// TIA Portal V16 export
// export: Created 2021-08-30T10:49:32.4865879Z, ExportSetting WithDefaults, DisplayName Totally Integrated Automation Portal, DisplayVersion V16 Update 3, DisplayName TIA Portal Version Control Interface, DisplayVersion V16 Update 2, DisplayName TIA Portal Openness, DisplayVersion V16 Update 3, DisplayName TIA Portal Teamcenter Gateway, DisplayVersion V16, DisplayName STEP 7 Professional, DisplayVersion V16 Update 3, DisplayName STEP 7 Safety, DisplayVersion V16, DisplayName WinCC Advanced, DisplayVersion V16 Update 3
FUNCTION_BLOCK "PumpCntrl2Pu1Fc"   // FB61, FBD
{ S7_Optimized_Access := 'TRUE' }
VERSION : 0.1
// 0 0 -стоп, 1- работа
// 1 2 - Запуск
// 2 4 - Остановка
// 3 8 - Сервисный режим
// 4 16 - Ошибка пуска
// 5 32 - Ошибка останова
// 6 64 - Ошибка питания
// 7 128 - Ошибка Частотника
// 8 256 - Блокировка внешняя (сборная)
// 9 - 512 - Нажат аварийный стоп
// 10 -U24 - Сборная авария
// 11 - 2048 - Местный режим
// 12 -  4096 - Ошибка вклчюния контактора
// 13 - 8192 - шбика отключения контактора
// 14 -  16384 - 1 показывать кнопки ручного управления
// 15 - 32768 - режим 1-ручной, 0-авто (только для индикатора на скаде)
// stored: AutoNumber false, IsIECCheckEnabled false, IsRetainMemResEnabled false, MemoryReserve 100, SetENOAutomatically false, UDAEnableTagReadback false
   VAR_INPUT
      modePU : Bool;
      cmPU : Bool;
      iWorkUZ : Bool;
      iAlarmFC : Bool;
      iKM1 : Bool;
      iKM2 : Bool;
      enableChange : Bool;
      Ack : Bool;
      blockPU1_1 : Bool;
      blockPU1_2 : Bool;
      blockPU1_3 : Bool;
      blockPU1_4 : Bool;
      blockPU1_5 : Bool;
      blockPU1_6 : Bool;
      blockPU1_7 : Bool;
      blockPU1_8 : Bool;
      blockPU2_1 : Bool;
      blockPU2_2 : Bool;
      blockPU2_3 : Bool;
      blockPU2_4 : Bool;
      blockPU2_5 : Bool;
      blockPU2_6 : Bool;
      blockPU2_7 : Bool;
      blockPU2_8 : Bool;
   END_VAR
   VAR_OUTPUT
      qKM_PU1 : Bool;
      qKM_PU2 : Bool;
      qUZ : Bool;
      showPU1_button : Bool;
      showPU2_button : Bool;
      tChangeRealHour : Real;
   END_VAR
   VAR_IN_OUT
      select : Bool;
      PU1 : "Pump";
      PU2 : "Pump";
   END_VAR
   VAR
      cmPU1 : Bool;   // Врутренняя команда первого насоса
      cmPU2 : Bool;   // Врутренняя команда второго насоса
      selectInternal : Bool;
      TOFcmPU1 { S7_SetPoint := 'True'} : TOF_TIME;
      TOFcmPU2 { S7_SetPoint := 'True'} : TOF_TIME;
   END_VAR
   VAR RETAIN
      tWork1 : DInt;
      tWork2 : DInt;
   END_VAR
   VAR
      tChange : DInt;
      needChange : Bool;
      tmpDInt : DInt;
      errAlarmFC_PU1 : Bool;
      errAlarmFC_PU2 : Bool;
      errBlock_PU1 : Bool;
      errBlock_PU2 : Bool;
      tmrErrOnUZ : TON_TIME;
      errON_UZ_PU1 : Bool;
      errON_UZ_PU2 : Bool;
      tmrErrOffUZ : TON_TIME;
      errOff_UZ_PU1 : Bool;
      errOff_UZ_PU2 : Bool;
      tmrErrOnKM_PU1 : TON_TIME;
      errOn_KM_PU1 : Bool;
      errOn_KM_PU2 : Bool;
      errOff_KM_PU1 : Bool;
      errOff_KM_PU2 : Bool;
      tmrErrOnKM_PU2 { S7_SetPoint := 'True'} : TON_TIME;
      tmrErrOffKM_PU1 { S7_SetPoint := 'True'} : TON_TIME;
      tmrErrOffKM_PU2 { S7_SetPoint := 'True'} : TON_TIME;
      errServicePU1 : Bool;
      errServicePU2 : Bool;
      tStartPU_FC : Time;
      tStopPU_FC : Time;
   END_VAR
BEGIN

REGION Network 1: Режим
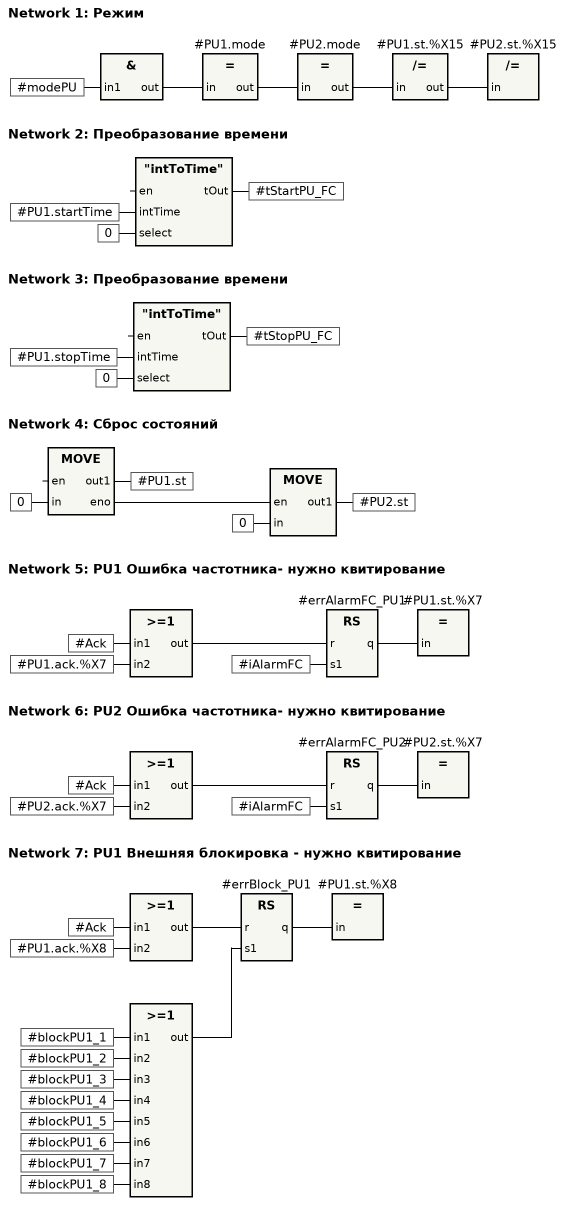
   #PU1.mode := #modePU;
   #PU2.mode := #modePU;
   #PU1.st.%X15 := NOT #modePU;
   #PU2.st.%X15 := NOT #modePU;
END_REGION

REGION Network 2: Преобразование времени
   // ВРемя из настроек первого насоса
   "intToTime"(intTime := #PU1.startTime, select := 0, tOut => #tStartPU_FC);
END_REGION

REGION Network 3: Преобразование времени
   // ВРемя из настроек первого насоса
   "intToTime"(intTime := #PU1.stopTime, select := 0, tOut => #tStopPU_FC);
END_REGION

REGION Network 4: Сброс состояний
   #PU1.st := 0;
   #PU2.st := 0;
END_REGION

REGION Network 5: PU1 Ошибка частотника- нужно квитирование
   IF #Ack OR #PU1.ack.%X7 THEN
       #errAlarmFC_PU1 := FALSE;   // RS flip-flop
   END_IF;
   IF #iAlarmFC THEN #errAlarmFC_PU1 := TRUE; END_IF;
   #PU1.st.%X7 := #errAlarmFC_PU1;
END_REGION

REGION Network 6: PU2 Ошибка частотника- нужно квитирование
   IF #Ack OR #PU2.ack.%X7 THEN
       #errAlarmFC_PU2 := FALSE;   // RS flip-flop
   END_IF;
   IF #iAlarmFC THEN #errAlarmFC_PU2 := TRUE; END_IF;
   #PU2.st.%X7 := #errAlarmFC_PU2;
END_REGION

REGION Network 7: PU1 Внешняя блокировка - нужно квитирование
   IF #Ack OR #PU1.ack.%X8 THEN
       #errBlock_PU1 := FALSE;   // RS flip-flop
   END_IF;
   IF #blockPU1_1 OR #blockPU1_2 OR #blockPU1_3 OR #blockPU1_4 OR #blockPU1_5 OR #blockPU1_6 OR #blockPU1_7 OR #blockPU1_8 THEN
       #errBlock_PU1 := TRUE;
   END_IF;
   #PU1.st.%X8 := #errBlock_PU1;
END_REGION

REGION Network 8: Детализация блокировок PU1
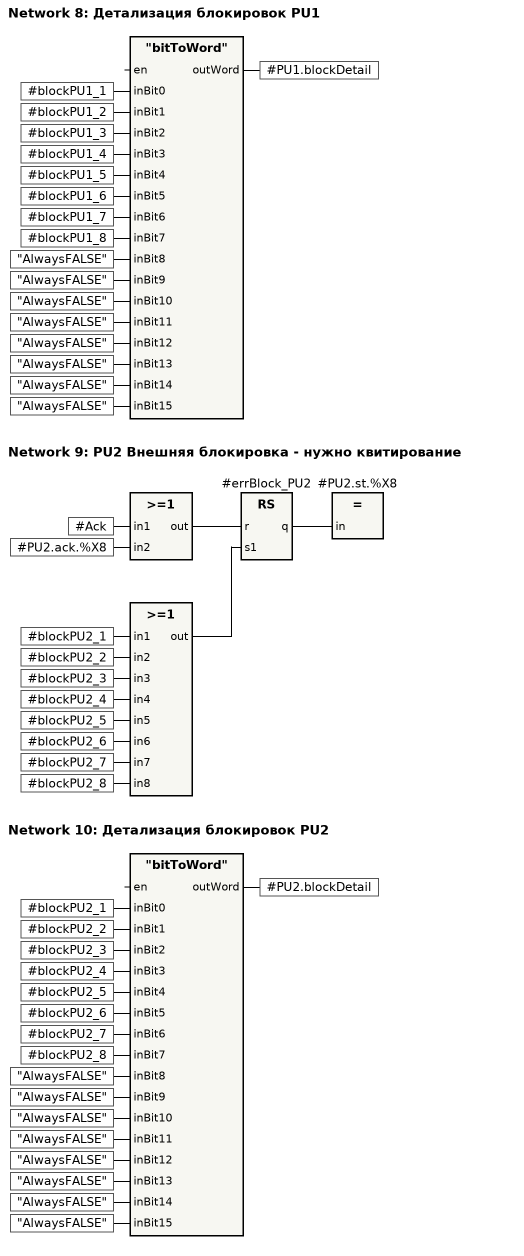
   "bitToWord"(inBit0 := #blockPU1_1,
               inBit1 := #blockPU1_2,
               inBit2 := #blockPU1_3,
               inBit3 := #blockPU1_4,
               inBit4 := #blockPU1_5,
               inBit5 := #blockPU1_6,
               inBit6 := #blockPU1_7,
               inBit7 := #blockPU1_8,
               inBit8 := "AlwaysFALSE",
               inBit9 := "AlwaysFALSE",
               inBit10 := "AlwaysFALSE",
               inBit11 := "AlwaysFALSE",
               inBit12 := "AlwaysFALSE",
               inBit13 := "AlwaysFALSE",
               inBit14 := "AlwaysFALSE",
               inBit15 := "AlwaysFALSE",
               outWord => #PU1.blockDetail);
END_REGION

REGION Network 9: PU2 Внешняя блокировка - нужно квитирование
   IF #Ack OR #PU2.ack.%X8 THEN
       #errBlock_PU2 := FALSE;   // RS flip-flop
   END_IF;
   IF #blockPU2_1 OR #blockPU2_2 OR #blockPU2_3 OR #blockPU2_4 OR #blockPU2_5 OR #blockPU2_6 OR #blockPU2_7 OR #blockPU2_8 THEN
       #errBlock_PU2 := TRUE;
   END_IF;
   #PU2.st.%X8 := #errBlock_PU2;
END_REGION

REGION Network 10: Детализация блокировок PU2
   "bitToWord"(inBit0 := #blockPU2_1,
               inBit1 := #blockPU2_2,
               inBit2 := #blockPU2_3,
               inBit3 := #blockPU2_4,
               inBit4 := #blockPU2_5,
               inBit5 := #blockPU2_6,
               inBit6 := #blockPU2_7,
               inBit7 := #blockPU2_8,
               inBit8 := "AlwaysFALSE",
               inBit9 := "AlwaysFALSE",
               inBit10 := "AlwaysFALSE",
               inBit11 := "AlwaysFALSE",
               inBit12 := "AlwaysFALSE",
               inBit13 := "AlwaysFALSE",
               inBit14 := "AlwaysFALSE",
               inBit15 := "AlwaysFALSE",
               outWord => #PU2.blockDetail);
END_REGION

REGION Network 11: таймер включения частотника
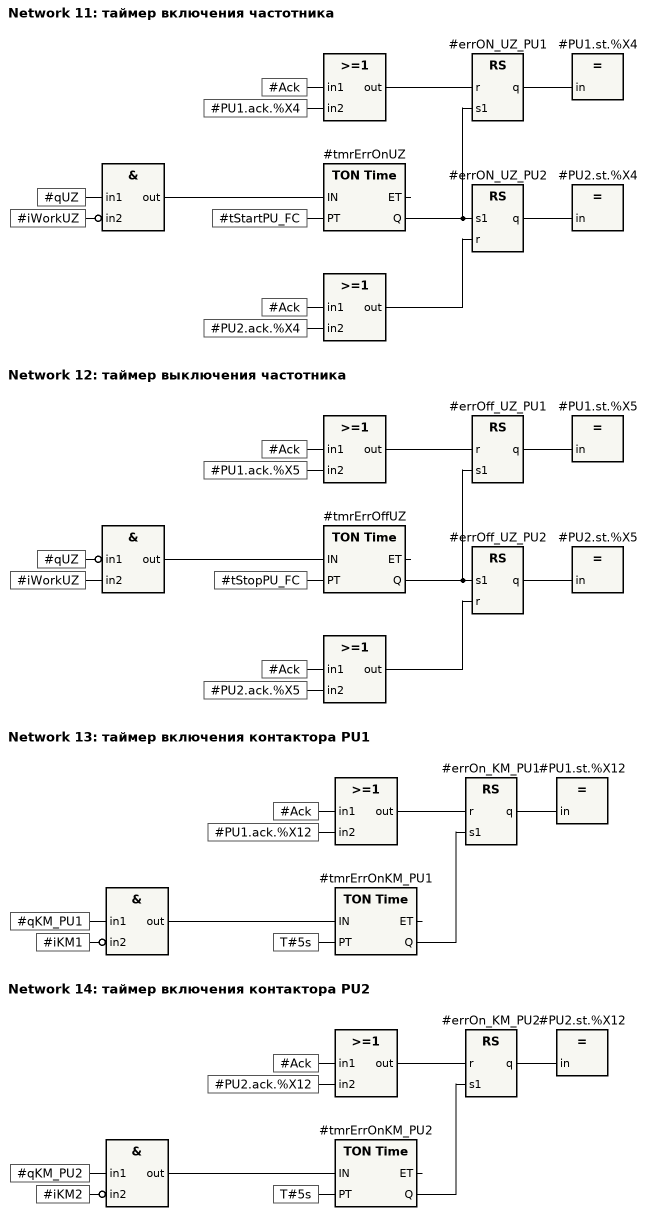
   #tmrErrOnUZ(IN := #qUZ AND NOT #iWorkUZ, PT := #tStartPU_FC);   // TON
   IF #Ack OR #PU1.ack.%X4 THEN
       #errON_UZ_PU1 := FALSE;   // RS flip-flop
   END_IF;
   IF #tmrErrOnUZ.Q THEN #errON_UZ_PU1 := TRUE; END_IF;
   #PU1.st.%X4 := #errON_UZ_PU1;
   IF #Ack OR #PU2.ack.%X4 THEN
       #errON_UZ_PU2 := FALSE;   // RS flip-flop
   END_IF;
   IF #tmrErrOnUZ.Q THEN #errON_UZ_PU2 := TRUE; END_IF;
   #PU2.st.%X4 := #errON_UZ_PU2;
END_REGION

REGION Network 12: таймер выключения частотника
   #tmrErrOffUZ(IN := NOT #qUZ AND #iWorkUZ, PT := #tStopPU_FC);   // TON
   IF #Ack OR #PU1.ack.%X5 THEN
       #errOff_UZ_PU1 := FALSE;   // RS flip-flop
   END_IF;
   IF #tmrErrOffUZ.Q THEN #errOff_UZ_PU1 := TRUE; END_IF;
   #PU1.st.%X5 := #errOff_UZ_PU1;
   IF #Ack OR #PU2.ack.%X5 THEN
       #errOff_UZ_PU2 := FALSE;   // RS flip-flop
   END_IF;
   IF #tmrErrOffUZ.Q THEN #errOff_UZ_PU2 := TRUE; END_IF;
   #PU2.st.%X5 := #errOff_UZ_PU2;
END_REGION

REGION Network 13: таймер включения контактора PU1
   #tmrErrOnKM_PU1(IN := #qKM_PU1 AND NOT #iKM1, PT := T#5s);   // TON
   IF #Ack OR #PU1.ack.%X12 THEN
       #errOn_KM_PU1 := FALSE;   // RS flip-flop
   END_IF;
   IF #tmrErrOnKM_PU1.Q THEN #errOn_KM_PU1 := TRUE; END_IF;
   #PU1.st.%X12 := #errOn_KM_PU1;
END_REGION

REGION Network 14: таймер включения контактора PU2
   #tmrErrOnKM_PU2(IN := #qKM_PU2 AND NOT #iKM2, PT := T#5s);   // TON
   IF #Ack OR #PU2.ack.%X12 THEN
       #errOn_KM_PU2 := FALSE;   // RS flip-flop
   END_IF;
   IF #tmrErrOnKM_PU2.Q THEN #errOn_KM_PU2 := TRUE; END_IF;
   #PU2.st.%X12 := #errOn_KM_PU2;
END_REGION

REGION Network 15: таймер отключения контактора PU1
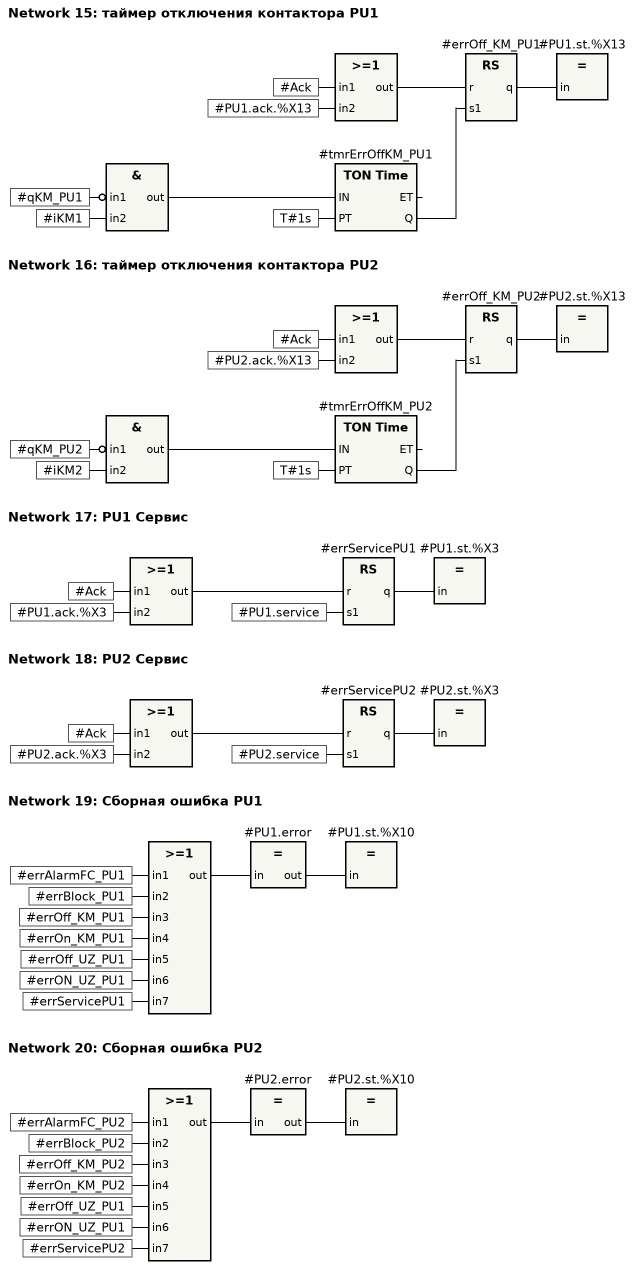
   #tmrErrOffKM_PU1(IN := NOT #qKM_PU1 AND #iKM1, PT := T#1s);   // TON
   IF #Ack OR #PU1.ack.%X13 THEN
       #errOff_KM_PU1 := FALSE;   // RS flip-flop
   END_IF;
   IF #tmrErrOffKM_PU1.Q THEN #errOff_KM_PU1 := TRUE; END_IF;
   #PU1.st.%X13 := #errOff_KM_PU1;
END_REGION

REGION Network 16: таймер отключения контактора PU2
   #tmrErrOffKM_PU2(IN := NOT #qKM_PU2 AND #iKM2, PT := T#1s);   // TON
   IF #Ack OR #PU2.ack.%X13 THEN
       #errOff_KM_PU2 := FALSE;   // RS flip-flop
   END_IF;
   IF #tmrErrOffKM_PU2.Q THEN #errOff_KM_PU2 := TRUE; END_IF;
   #PU2.st.%X13 := #errOff_KM_PU2;
END_REGION

REGION Network 17: PU1 Сервис
   IF #Ack OR #PU1.ack.%X3 THEN
       #errServicePU1 := FALSE;   // RS flip-flop
   END_IF;
   IF #PU1.service THEN #errServicePU1 := TRUE; END_IF;
   #PU1.st.%X3 := #errServicePU1;
END_REGION

REGION Network 18: PU2 Сервис
   IF #Ack OR #PU2.ack.%X3 THEN
       #errServicePU2 := FALSE;   // RS flip-flop
   END_IF;
   IF #PU2.service THEN #errServicePU2 := TRUE; END_IF;
   #PU2.st.%X3 := #errServicePU2;
END_REGION

REGION Network 19: Сборная ошибка РU1
   #PU1.error := #errAlarmFC_PU1 OR #errBlock_PU1 OR #errOff_KM_PU1 OR #errOn_KM_PU1 OR #errOff_UZ_PU1 OR #errON_UZ_PU1 OR #errServicePU1;
   #PU1.st.%X10 := #PU1.error;
END_REGION

REGION Network 20: Сборная ошибка РU2
   #PU2.error := #errAlarmFC_PU2 OR #errBlock_PU2 OR #errOff_KM_PU2 OR #errOn_KM_PU2 OR #errOff_UZ_PU1 OR #errON_UZ_PU1 OR #errServicePU2;
   #PU2.st.%X10 := #PU2.error;
END_REGION

REGION Network 21: Состояние работает PU1
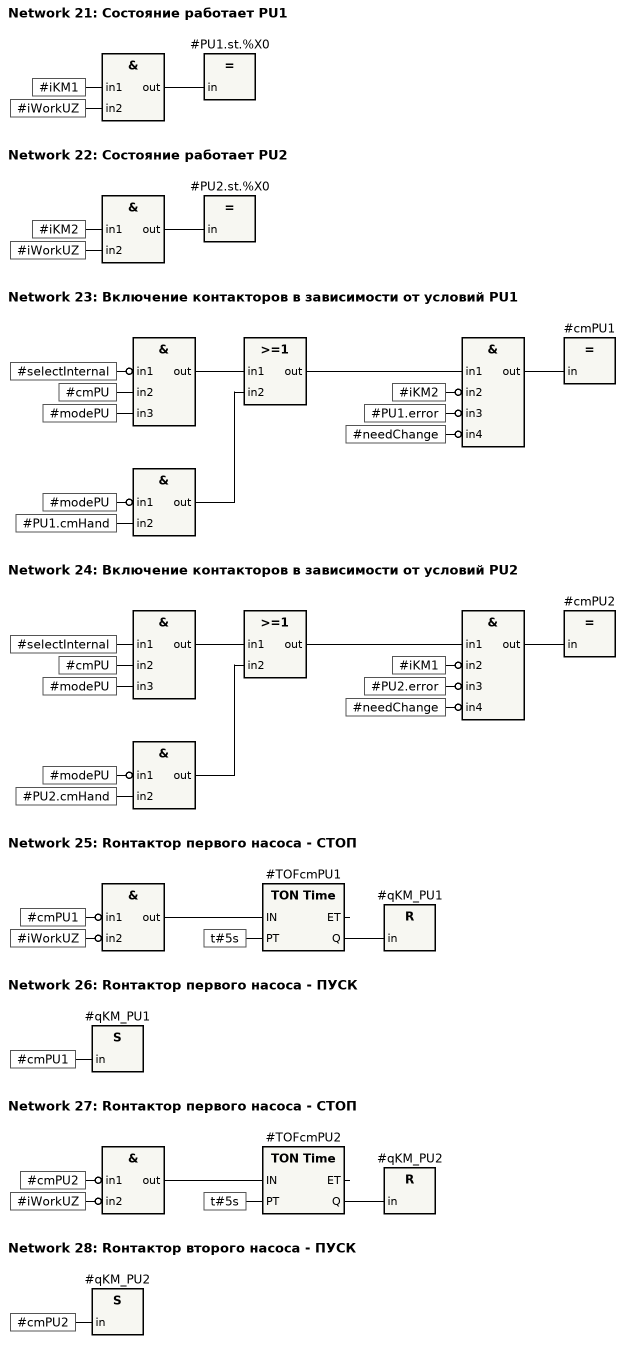
   #PU1.st.%X0 := #iKM1 AND #iWorkUZ;
END_REGION

REGION Network 22: Состояние работает PU2
   #PU2.st.%X0 := #iKM2 AND #iWorkUZ;
END_REGION

REGION Network 23: Включение контакторов в зависимости от условий PU1
   #cmPU1 := ((NOT #selectInternal AND #cmPU AND #modePU) OR (NOT #modePU AND #PU1.cmHand)) AND NOT #iKM2 AND NOT #PU1.error AND NOT #needChange;
END_REGION

REGION Network 24: Включение контакторов в зависимости от условий PU2
   #cmPU2 := ((#selectInternal AND #cmPU AND #modePU) OR (NOT #modePU AND #PU2.cmHand)) AND NOT #iKM1 AND NOT #PU2.error AND NOT #needChange;
END_REGION

REGION Network 25: Rонтактор первого насоса - СТОП
   #TOFcmPU1(IN := NOT #cmPU1 AND NOT #iWorkUZ, PT := t#5s);   // TON
   IF #TOFcmPU1.Q THEN #qKM_PU1 := FALSE; END_IF;
END_REGION

REGION Network 26: Rонтактор первого насоса - ПУСК
   IF #cmPU1 THEN #qKM_PU1 := TRUE; END_IF;
END_REGION

REGION Network 27: Rонтактор первого насоса - СТОП
   #TOFcmPU2(IN := NOT #cmPU2 AND NOT #iWorkUZ, PT := t#5s);   // TON
   IF #TOFcmPU2.Q THEN #qKM_PU2 := FALSE; END_IF;
END_REGION

REGION Network 28: Rонтактор второго насоса - ПУСК
   IF #cmPU2 THEN #qKM_PU2 := TRUE; END_IF;
END_REGION

REGION Network 29: Команда на UZ
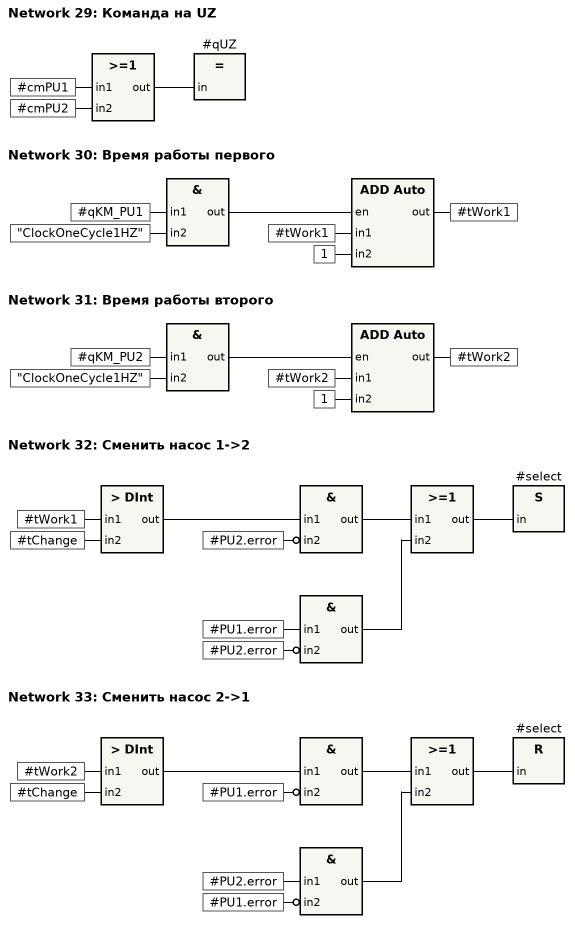
   #qUZ := #cmPU1 OR #cmPU2;
END_REGION

REGION Network 30: Время работы первого
   IF #qKM_PU1 AND "ClockOneCycle1HZ" THEN #tWork1 := #tWork1 + 1; END_IF;
END_REGION

REGION Network 31: Время работы второго
   IF #qKM_PU2 AND "ClockOneCycle1HZ" THEN #tWork2 := #tWork2 + 1; END_IF;
END_REGION

REGION Network 32: Сменить насос 1->2
   IF ((#tWork1 > #tChange) AND NOT #PU2.error) OR (#PU1.error AND NOT #PU2.error) THEN
       #select := TRUE;
   END_IF;
END_REGION

REGION Network 33: Сменить насос 2->1
   IF ((#tWork2 > #tChange) AND NOT #PU1.error) OR (#PU2.error AND NOT #PU1.error) THEN
       #select := FALSE;
   END_IF;
END_REGION

REGION Network 34
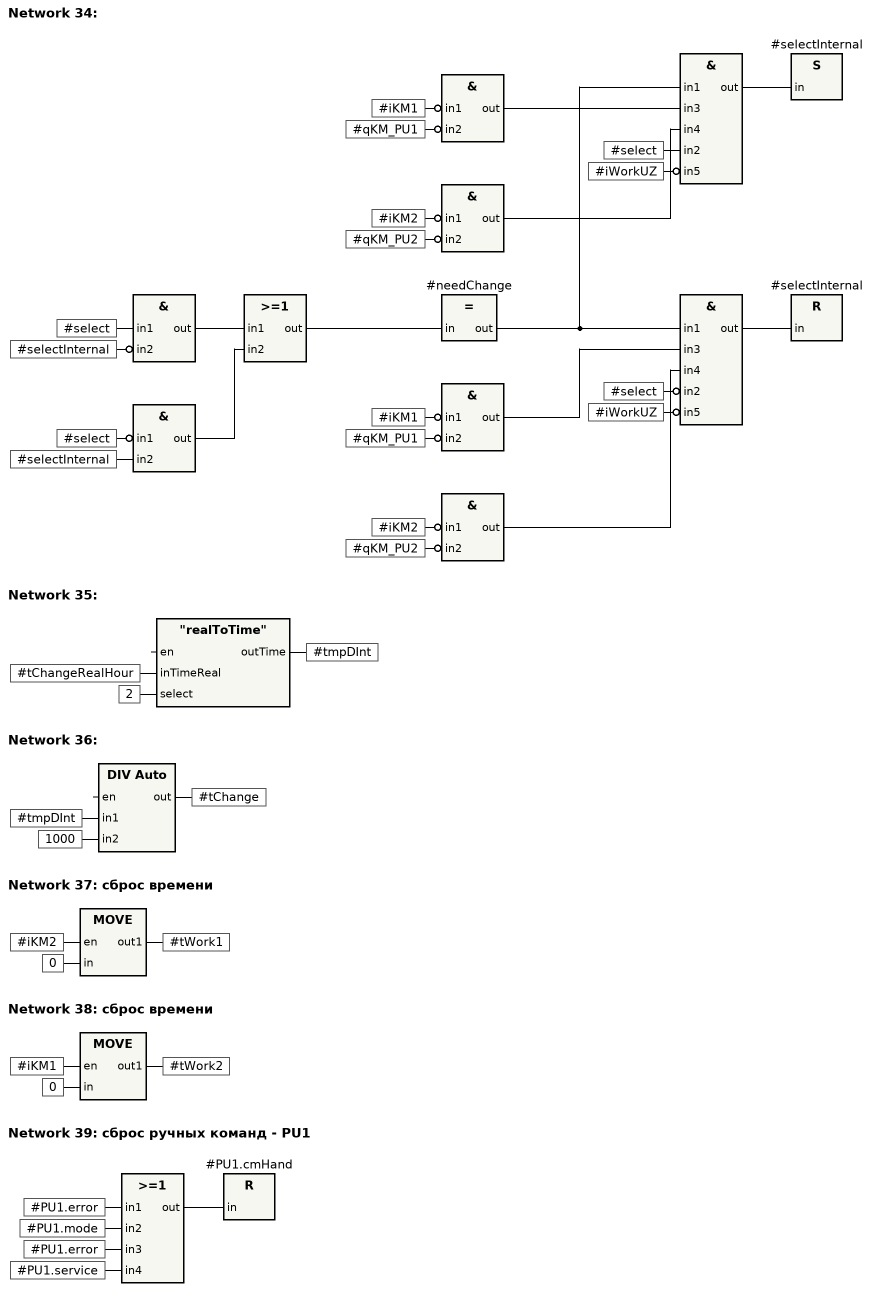
   #needChange := (#select AND NOT #selectInternal) OR (NOT #select AND #selectInternal);
   IF #needChange AND NOT #iKM1 AND NOT #qKM_PU1 AND NOT #iKM2 AND NOT #qKM_PU2 AND #select AND NOT #iWorkUZ THEN
       #selectInternal := TRUE;
   END_IF;
   IF #needChange AND NOT #iKM1 AND NOT #qKM_PU1 AND NOT #iKM2 AND NOT #qKM_PU2 AND NOT #select AND NOT #iWorkUZ THEN
       #selectInternal := FALSE;
   END_IF;
END_REGION

REGION Network 35
   "realToTime"(inTimeReal := #tChangeRealHour, select := 2, outTime => #tmpDInt);
END_REGION

REGION Network 36
   #tChange := #tmpDInt / 1000;
END_REGION

REGION Network 37: сброс времени
   IF #iKM2 THEN #tWork1 := 0; END_IF;
END_REGION

REGION Network 38: сброс времени
   IF #iKM1 THEN #tWork2 := 0; END_IF;
END_REGION

REGION Network 39: сброс ручных команд - PU1
   IF #PU1.error OR #PU1.mode OR #PU1.error OR #PU1.service THEN #PU1.cmHand := FALSE; END_IF;
END_REGION

REGION Network 40: ручная команда - PU2
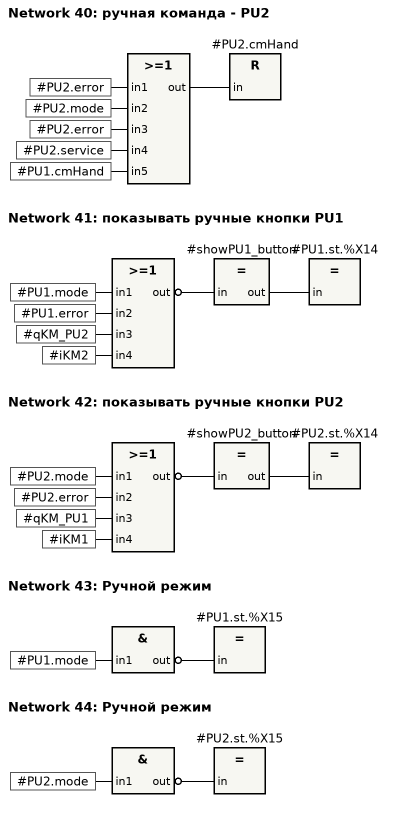
   IF #PU2.error OR #PU2.mode OR #PU2.error OR #PU2.service OR #PU1.cmHand THEN #PU2.cmHand := FALSE; END_IF;
END_REGION

REGION Network 41: показывать ручные кнопки PU1
   #showPU1_button := NOT (#PU1.mode OR #PU1.error OR #qKM_PU2 OR #iKM2);
   #PU1.st.%X14 := #showPU1_button;
END_REGION

REGION Network 42: показывать ручные кнопки PU2
   #showPU2_button := NOT (#PU2.mode OR #PU2.error OR #qKM_PU1 OR #iKM1);
   #PU2.st.%X14 := #showPU2_button;
END_REGION

REGION Network 43: Ручной режим
   #PU1.st.%X15 := NOT #PU1.mode;
END_REGION

REGION Network 44: Ручной режим
   #PU2.st.%X15 := NOT #PU2.mode;
END_REGION

REGION Network 45 (SCL): Сброс битов Ack
   IF NOT #PU1.st.%X0 AND #PU1.ack.%X0 THEN
       #PU1.ack.%X0 := 0;
   END_IF;
   IF NOT #PU1.st.%X1 AND #PU1.ack.%X1 THEN
       #PU1.ack.%X1 := 0;
   END_IF;
   IF NOT #PU1.st.%X2 AND #PU1.ack.%X2 THEN
       #PU1.ack.%X2 := 0;
   END_IF;
   IF NOT #PU1.st.%X3 AND #PU1.ack.%X3 THEN
       #PU1.ack.%X3 := 0;
   END_IF;
   IF NOT #PU1.st.%X4 AND #PU1.ack.%X4 THEN
       #PU1.ack.%X4 := 0;
   END_IF;
   IF NOT #PU1.st.%X5 AND #PU1.ack.%X5 THEN
       #PU1.ack.%X5 := 0;
   END_IF;
   IF NOT #PU1.st.%X6 AND #PU1.ack.%X6 THEN
       #PU1.ack.%X6 := 0;
   END_IF;
   IF NOT #PU1.st.%X7 AND #PU1.ack.%X7 THEN
       #PU1.ack.%X7 := 0;
   END_IF;
   IF NOT #PU1.st.%X8 AND #PU1.ack.%X8 THEN
       #PU1.ack.%X8 := 0;
   END_IF;
   IF NOT #PU1.st.%X9 AND #PU1.ack.%X9 THEN
       #PU1.ack.%X9 := 0;
   END_IF;
   IF NOT #PU1.st.%X10 AND #PU1.ack.%X10 THEN
       #PU1.ack.%X10 := 0;
   END_IF;
   IF NOT #PU1.st.%X11 AND #PU1.ack.%X11 THEN
       #PU1.ack.%X11 := 0;
   END_IF;
   IF NOT #PU1.st.%X12 AND #PU1.ack.%X12 THEN
       #PU1.ack.%X12 := 0;
   END_IF;
   IF NOT #PU1.st.%X13 AND #PU1.ack.%X13 THEN
       #PU1.ack.%X13 := 0;
   END_IF;
   IF NOT #PU1.st.%X14 AND #PU1.ack.%X14 THEN
       #PU1.ack.%X14 := 0;
   END_IF;
   IF NOT #PU1.st.%X15 AND #PU1.ack.%X15 THEN
       #PU1.ack.%X15 := 0;
   END_IF;
   IF NOT #PU2.st.%X0 AND #PU2.ack.%X0 THEN
       #PU2.ack.%X0 := 0;
   END_IF;
   IF NOT #PU2.st.%X1 AND #PU2.ack.%X1 THEN
       #PU2.ack.%X1 := 0;
   END_IF;
   IF NOT #PU2.st.%X2 AND #PU2.ack.%X2 THEN
       #PU2.ack.%X2 := 0;
   END_IF;
   IF NOT #PU2.st.%X3 AND #PU2.ack.%X3 THEN
       #PU2.ack.%X3 := 0;
   END_IF;
   IF NOT #PU2.st.%X4 AND #PU2.ack.%X4 THEN
       #PU2.ack.%X4 := 0;
   END_IF;
   IF NOT #PU2.st.%X5 AND #PU2.ack.%X5 THEN
       #PU2.ack.%X5 := 0;
   END_IF;
   IF NOT #PU2.st.%X6 AND #PU2.ack.%X6 THEN
       #PU2.ack.%X6 := 0;
   END_IF;
   IF NOT #PU2.st.%X7 AND #PU2.ack.%X7 THEN
       #PU2.ack.%X7 := 0;
   END_IF;
   IF NOT #PU2.st.%X8 AND #PU2.ack.%X8 THEN
       #PU2.ack.%X8 := 0;
   END_IF;
   IF NOT #PU2.st.%X9 AND #PU2.ack.%X9 THEN
       #PU2.ack.%X9 := 0;
   END_IF;
   IF NOT #PU2.st.%X10 AND #PU2.ack.%X10 THEN
       #PU2.ack.%X10 := 0;
   END_IF;
   IF NOT #PU2.st.%X11 AND #PU2.ack.%X11 THEN
       #PU2.ack.%X11 := 0;
   END_IF;
   IF NOT #PU2.st.%X12 AND #PU2.ack.%X12 THEN
       #PU2.ack.%X12 := 0;
   END_IF;
   IF NOT #PU2.st.%X13 AND #PU2.ack.%X13 THEN
       #PU2.ack.%X13 := 0;
   END_IF;
   IF NOT #PU2.st.%X14 AND #PU2.ack.%X14 THEN
       #PU2.ack.%X14 := 0;
   END_IF;
   IF NOT #PU2.st.%X15 AND #PU2.ack.%X15 THEN
       #PU2.ack.%X15 := 0;
   END_IF;
END_REGION
END_FUNCTION_BLOCK
